PROGRAM SafetyLogic
VAR
	SafetyRun AT %Q* : BOOL;
	ErrorActknowledgement AT %Q* : BOOL;
	ResetSafety AT %Q* : BOOL;
	TestOut1 AT %Q* : BOOL;
	TestIn1 AT %I* : BOOL;
	TurnOff AT %Q*  : BOOL;
END_VAR

SafetyRun := TRUE;

END_PROGRAM

(* stored: Version 1.1.0.1, ProductVersion 3.1.4024.12
   POU SafetyLogic: Id {4b752a0c-d853-4d91-8492-d0fdf9872ce3}, SpecialFunc None *)
